TYPE CyclicAxis_Input_typ :
	STRUCT
		Command 	: CyclicAxis_CMD_typ ;
		Parameter	: CyclicAxis_Param_typ ;
	END_STRUCT
END_TYPE

(* stored: Version 1.1.0.1, ProductVersion 3.1.4024.3
   DUT CyclicAxis_Input_typ: Id {30ea196f-27b5-058c-3bb5-5c2e6d5f25b5} *)
